Yaskawa INFORM job: FRONT_WELD_90ST-2_5240.JBI

/JOB
//NAME FRONT_WELD_90ST-2_5240
///FOLDERNAME 02-SKRZYNIE_JOBS
//POS
///NPOS 19,19,0,4,0,0
///TOOL 0
///POSTYPE PULSE
///PULSE
C00000=0,-52278,40443,0,6873,1
C00001=0,-52278,40443,5610,-49281,-70968
C00002=0,-42686,23640,7425,-34877,-79161
C00003=-14116,-58141,-26117,-21696,-5351,-66126
C00004=-47175,-26068,-21336,-663,15689,-73543
C00005=-43679,-19706,-10978,-10022,13573,-68879
C00006=-43586,-19780,-11053,-10056,13586,-68800
C00007=-35860,-24949,-16233,-12945,14700,-62445
C00008=-13769,-29473,-19781,-48598,22018,-43228
C00009=-14906,-39722,-32778,-45263,22245,-44952
C00010=-3902,-39042,-32149,-3317,17100,-71988
C00011=-3902,-39042,-32149,-3317,17100,-71988
C00012=-4516,-35765,-28109,-2071,17670,-72647
C00013=-4247,-35775,-28088,-2606,17639,-72371
C00014=27559,-32679,-25102,-47227,27630,-48538
C00015=42160,-28234,-21597,-54805,35918,-43754
C00016=48063,-35826,-27915,-64657,37344,-38904
C00017=24039,-44019,6278,-32369,22109,-19464
C00018=0,-52278,40443,0,6873,1
BC00000=805481
BC00001=805481
BC00002=933762
BC00003=982336
BC00004=1012002
BC00005=1012002
BC00006=1012002
BC00007=1012002
BC00008=1012002
BC00009=1012002
BC00010=1011676
BC00011=1011676
BC00012=1011676
BC00013=1011676
BC00014=1011676
BC00015=1011676
BC00016=1011676
BC00017=908673
BC00018=805481
///POSTYPE BASE
///RECTAN
///RCONF 0,0,0,0,0,0,0,0,0,0,0,0,0,0,0,0,0,0,0,0,0,0,0,0
P00501=-2.026,0.009,3.534,0.0000,0.0000,0.0000
///RCONF 1,0,0,0,0,0,0,0,0,0,0,0,0,0,0,0,0,0,0,0,0,0,0,0
P00502=-2.023,0.001,1.732,0.0000,0.0000,0.0000
P00503=0.138,-0.044,1.539,0.0000,0.0000,0.0000
P00504=-0.309,-0.010,1.636,0.0000,0.0000,0.0000
//INST
///DATE 2024/05/18 20:39
///ATTR SC,RW
///GROUP1 RB1,BS1
NOP
MOVJ C00000 BC00000 VJ=50.00
MOVJ C00001 BC00001 VJ=50.00
MOVJ C00002 BC00002 VJ=50.00
MOVJ C00003 BC00003 VJ=50.00
'::::::::::::::::::::::::::::::::
'W56
'::::::::::::::::::::::::::::::::
MOVL C00004 BC00004 V=666.7
SFTON P0501
MACRO1 MJ#(0) ARGF14
MOVL C00005 BC00005 V=166.7 PL=0
ARCON
MOVC C00006 BC00006 V=9.5
MOVC C00007 BC00007 V=9.5
SFTOF
SFTON P0502
MOVC C00008 BC00008 V=9.5
ARCOF
MOVL C00009 BC00009 V=333.3
SFTOF
MOVL C00010 BC00010 V=333.3
'::::::::::::::::::::::::::::::::
'W21
'::::::::::::::::::::::::::::::::
MOVL C00011 BC00011 V=166.7
SFTON P0503
MACRO1 MJ#(0) ARGF14
MOVL C00012 BC00012 V=166.7 PL=0
ARCON
MOVC C00013 BC00013 V=9.5
SFTOF
SFTON P0504
MOVC C00014 BC00014 V=9.5
MOVC C00015 BC00015 V=9.5
ARCOF
MOVL C00016 BC00016 V=250.0
SFTOF
MOVJ C00017 BC00017 VJ=50.00
MOVJ C00018 BC00018 VJ=50.00
END
